Omron CX-Programmer project NewProject (CX-Programmer 9.73)

# PLC NewPLC1: CP2E-N N

## Global symbols (name address type ; comment)
0.00 BOOL  ; CR MASTER ON
0.01 BOOL  ; EMERGENCY STOP
0.02 BOOL  ; AUT: 1 / MAN: 0
0.03 BOOL  ; PB START AUTO
0.04 BOOL  ; PB RESET
0.05 BOOL  ; PB ROBOT RUN INSPECTION
0.06 BOOL  ; PB CLAMP
0.07 BOOL  ; PB UNCLAMP
0.08 BOOL  ; RS UNCLAMP 1
0.09 BOOL  ; RS UNCLAMP 2
0.10 BOOL  ; RS CLAMP 1
0.11 BOOL  ; RS CLAMP 2
100.00 BOOL  ; CR SOL CLAMP
100.01 BOOL  ; CR SOL UNCLAMP
100.02 BOOL  ; LAMP PLC RUN
100.03 BOOL  ; LAMP FAULT & TL RED
100.04 BOOL  ; LAMP HOMEPOST & TL GREEN
100.05 BOOL  ; LAMP AUTO RUN & TL YELLOW
100.06 BOOL  ; BUZZER
100.07 BOOL  ; LAMP ROBOT RUN
101.00 BOOL  ; TL INSPECTION OK
101.01 BOOL  ; TL INSPECTION NG
101.02 BOOL  ; TL INSPECTION RUN
10.00 BOOL  ; MASTER ON
10.01 BOOL  ; MASTER OFF
10.02 BOOL  ; MANUAL MODE CONFIRM
10.03 BOOL  ; AUTO MODE CONFIRM
10.04 BOOL  ; FAULT CONFIRM
10.05 BOOL  ; ROBOT ERROR
1.00 BOOL  ; PHS AGV
30.00 BOOL  ; IR CR UNCLAMP
30.01 BOOL  ; IR CR CLAMP
50.00 BOOL  ; AUTO UNCLAMP HOMING
50.01 BOOL  ; AUTO CLAMP
50.02 BOOL  ; AUTO ROBOT START INSPECTION
90.00 BOOL  ; MAN UNCLAMP
90.01 BOOL  ; MAN CLAMP
90.02 BOOL  ; MAN ROBOT START INSPECTION
T000 BOOL  ; DELAY RESET SEQ
T001 BOOL  ; DELAY AGV IN
W1 CHANNEL  ; ROBOT STATE
W2 CHANNEL  ; INSPECTION RESULT
W3 CHANNEL  ; ROBOT ERROR STATUS
W4 CHANNEL  ; ROBOT PROJECT STATUS
W5 CHANNEL  ; PLC ON STATUS
W6 CHANNEL  ; FLAG BARCODE FAIL

## Program NewProgram1 (cyclic task 0)

### Section MAIN_PROGRAM

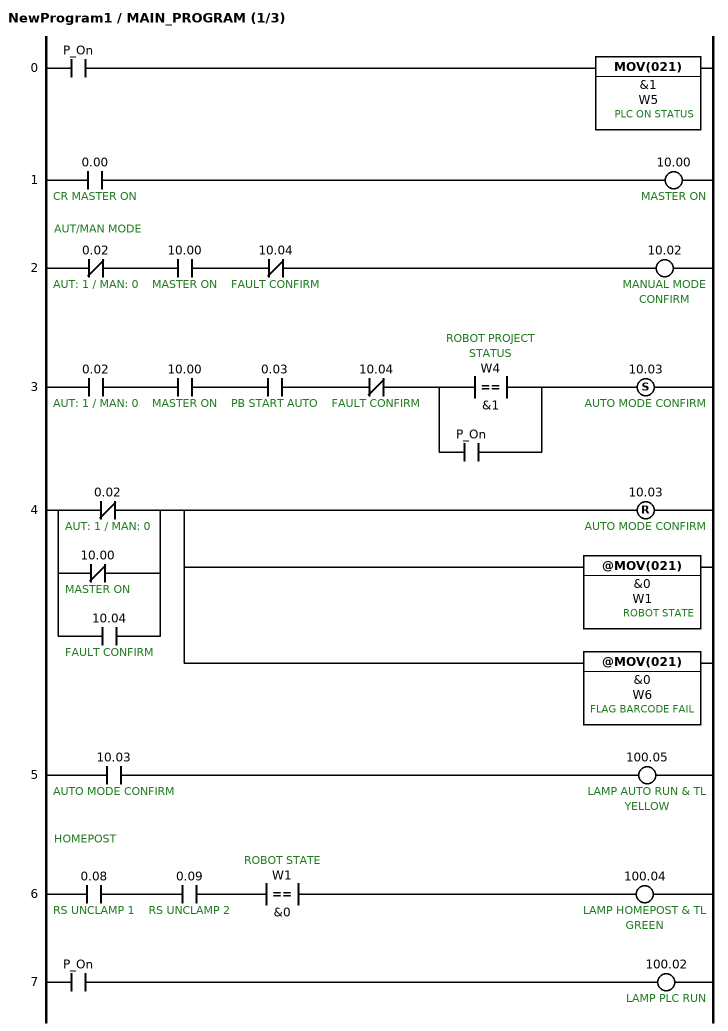
; rung 0
LD P_On
MOV(021) &1 W5  ; PLC ON STATUS
; rung 1
LD 0.00  ; CR MASTER ON
OUT 10.00  ; MASTER ON
; rung 2: AUT/MAN MODE
LDNOT 0.02  ; AUT: 1 / MAN: 0
AND 10.00  ; MASTER ON
ANDNOT 10.04  ; FAULT CONFIRM
OUT 10.02  ; MANUAL MODE CONFIRM
; rung 3
LD 0.02  ; AUT: 1 / MAN: 0
AND 10.00  ; MASTER ON
AND 0.03  ; PB START AUTO
ANDNOT 10.04  ; FAULT CONFIRM
LD=(300) W4 &1  ; ROBOT PROJECT STATUS
OR P_On
ANDLD
SET 10.03  ; AUTO MODE CONFIRM
; rung 4
LDNOT 0.02  ; AUT: 1 / MAN: 0
ORNOT 10.00  ; MASTER ON
OR 10.04  ; FAULT CONFIRM
RSET 10.03  ; AUTO MODE CONFIRM
@MOV(021) &0 W1  ; ROBOT STATE
@MOV(021) &0 W6  ; FLAG BARCODE FAIL
; rung 5
LD 10.03  ; AUTO MODE CONFIRM
OUT 100.05  ; LAMP AUTO RUN & TL YELLOW
; rung 6: HOMEPOST
LD 0.08  ; RS UNCLAMP 1
AND 0.09  ; RS UNCLAMP 2
AND=(300) W1 &0  ; ROBOT STATE
OUT 100.04  ; LAMP HOMEPOST & TL GREEN
; rung 7
LD P_On
OUT 100.02  ; LAMP PLC RUN

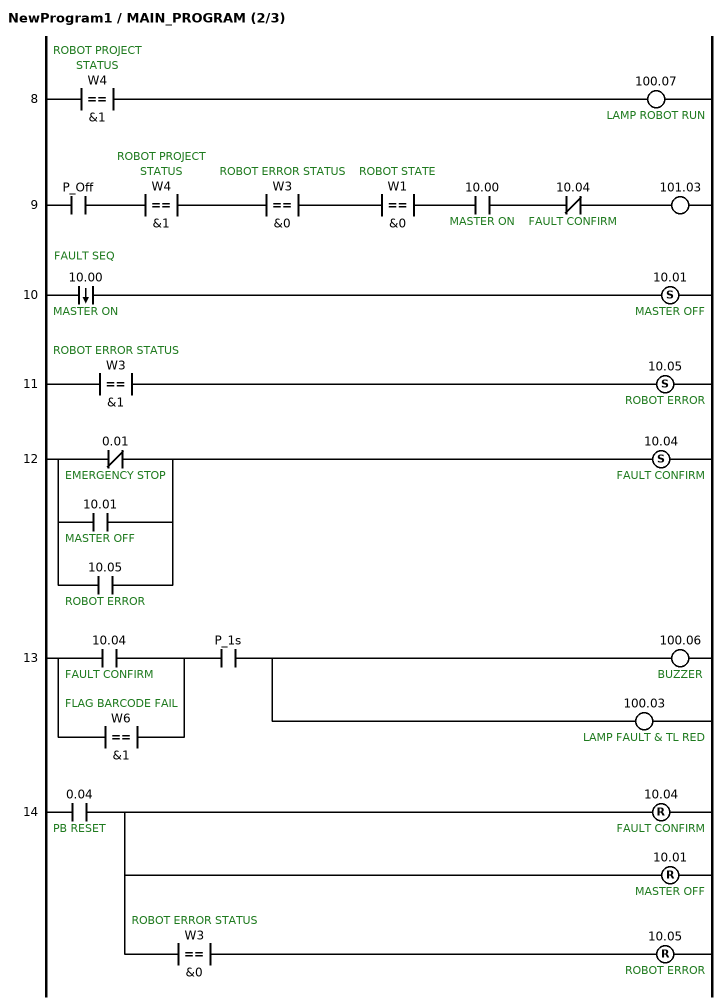
; rung 8
LD=(300) W4 &1  ; ROBOT PROJECT STATUS
OUT 100.07  ; LAMP ROBOT RUN
; rung 9
LD P_Off
AND=(300) W4 &1  ; ROBOT PROJECT STATUS
AND=(300) W3 &0  ; ROBOT ERROR STATUS
AND=(300) W1 &0  ; ROBOT STATE
AND 10.00  ; MASTER ON
ANDNOT 10.04  ; FAULT CONFIRM
OUT 101.03
; rung 10: FAULT SEQ
%LD 10.00  ; MASTER ON
SET 10.01  ; MASTER OFF
; rung 11
LD=(300) W3 &1  ; ROBOT ERROR STATUS
SET 10.05  ; ROBOT ERROR
; rung 12
LDNOT 0.01  ; EMERGENCY STOP
OR 10.01  ; MASTER OFF
OR 10.05  ; ROBOT ERROR
SET 10.04  ; FAULT CONFIRM
; rung 13
LD 10.04  ; FAULT CONFIRM
OR=(300) W6 &1  ; FLAG BARCODE FAIL
AND P_1s
OUT 100.06  ; BUZZER
OUT 100.03  ; LAMP FAULT & TL RED
; rung 14
LD 0.04  ; PB RESET
RSET 10.04  ; FAULT CONFIRM
RSET 10.01  ; MASTER OFF
AND=(300) W3 &0  ; ROBOT ERROR STATUS
RSET 10.05  ; ROBOT ERROR

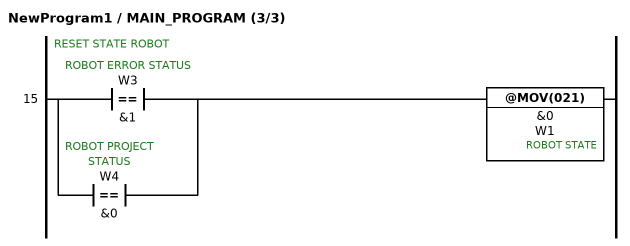
; rung 15: RESET STATE ROBOT
LD=(300) W3 &1  ; ROBOT ERROR STATUS
OR=(300) W4 &0  ; ROBOT PROJECT STATUS
@MOV(021) &0 W1  ; ROBOT STATE

### Section MANUAL

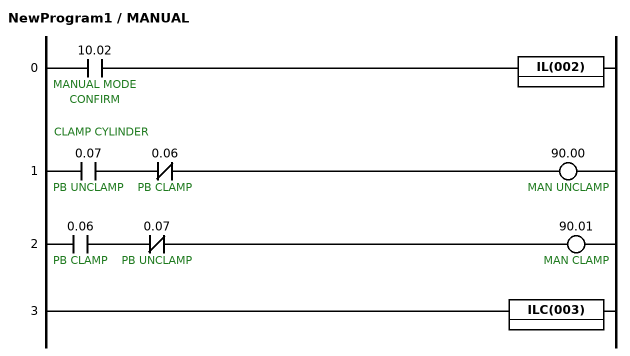
; rung 0
LD 10.02  ; MANUAL MODE CONFIRM
IL(002)
; rung 1: CLAMP CYLINDER
LD 0.07  ; PB UNCLAMP
ANDNOT 0.06  ; PB CLAMP
OUT 90.00  ; MAN UNCLAMP
; rung 2
LD 0.06  ; PB CLAMP
ANDNOT 0.07  ; PB UNCLAMP
OUT 90.01  ; MAN CLAMP
; rung 3
ILC(003)

### Section AUTO

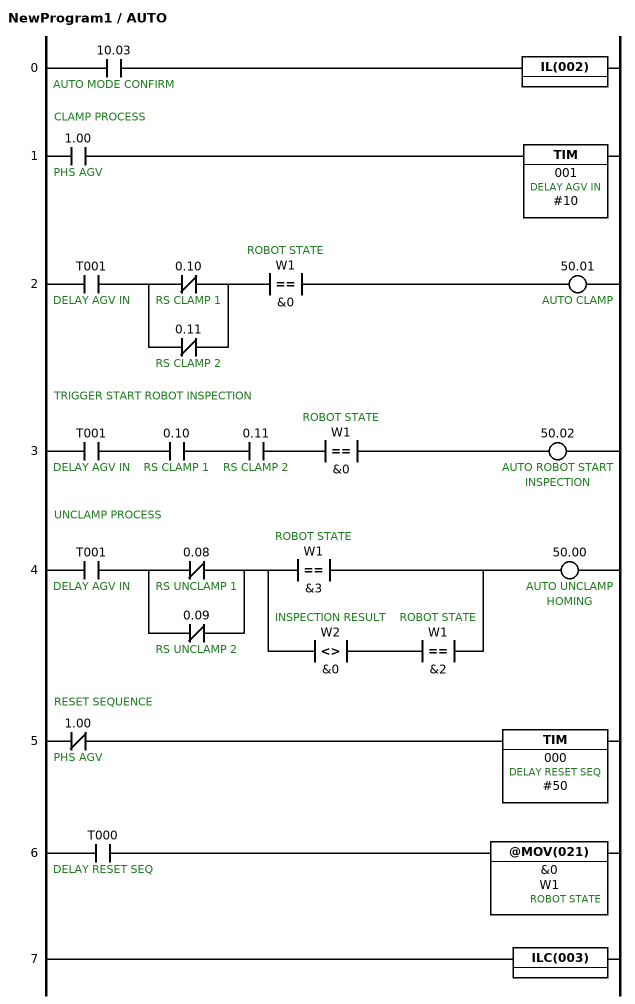
; rung 0
LD 10.03  ; AUTO MODE CONFIRM
IL(002)
; rung 1: CLAMP PROCESS
LD 1.00  ; PHS AGV
TIM 001 #10  ; DELAY AGV IN
; rung 2
LD T001  ; DELAY AGV IN
LDNOT 0.10  ; RS CLAMP 1
ORNOT 0.11  ; RS CLAMP 2
ANDLD
AND=(300) W1 &0  ; ROBOT STATE
OUT 50.01  ; AUTO CLAMP
; rung 3: TRIGGER START ROBOT INSPECTION
LD T001  ; DELAY AGV IN
AND 0.10  ; RS CLAMP 1
AND 0.11  ; RS CLAMP 2
AND=(300) W1 &0  ; ROBOT STATE
OUT 50.02  ; AUTO ROBOT START INSPECTION
; rung 4: UNCLAMP PROCESS
LD T001  ; DELAY AGV IN
LDNOT 0.08  ; RS UNCLAMP 1
ORNOT 0.09  ; RS UNCLAMP 2
ANDLD
LD=(300) W1 &3  ; ROBOT STATE
LD<>(305) W2 &0  ; INSPECTION RESULT
AND=(300) W1 &2  ; ROBOT STATE
ORLD
ANDLD
OUT 50.00  ; AUTO UNCLAMP HOMING
; rung 5: RESET SEQUENCE
LDNOT 1.00  ; PHS AGV
TIM 000 #50  ; DELAY RESET SEQ
; rung 6
LD T000  ; DELAY RESET SEQ
@MOV(021) &0 W1  ; ROBOT STATE
; rung 7
ILC(003)

### Section OUTPUT

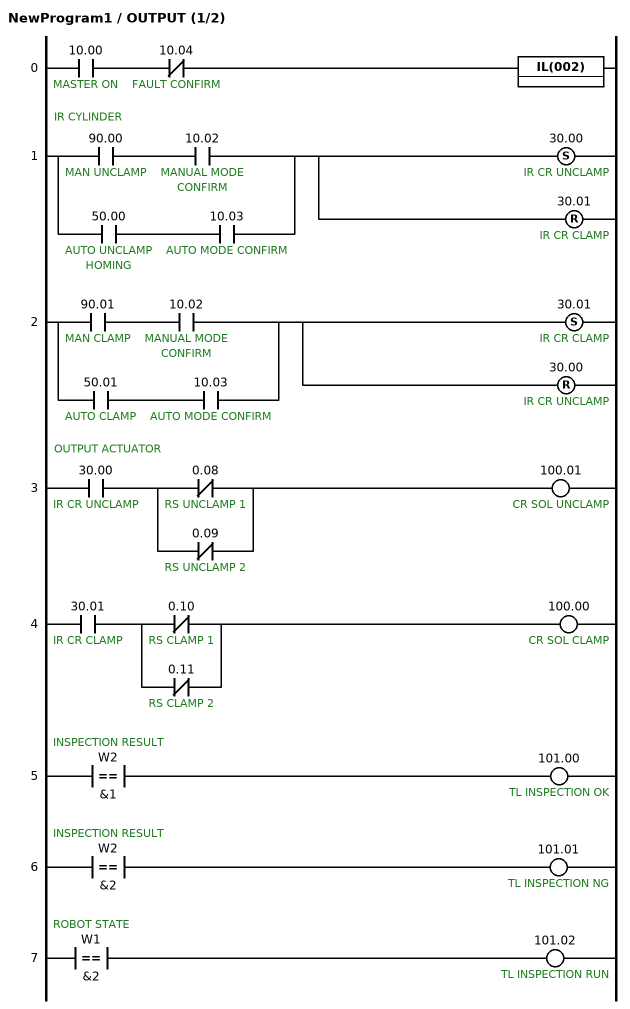
; rung 0
LD 10.00  ; MASTER ON
ANDNOT 10.04  ; FAULT CONFIRM
IL(002)
; rung 1: IR CYLINDER
LD 90.00  ; MAN UNCLAMP
AND 10.02  ; MANUAL MODE CONFIRM
LD 50.00  ; AUTO UNCLAMP HOMING
AND 10.03  ; AUTO MODE CONFIRM
ORLD
SET 30.00  ; IR CR UNCLAMP
RSET 30.01  ; IR CR CLAMP
; rung 2
LD 90.01  ; MAN CLAMP
AND 10.02  ; MANUAL MODE CONFIRM
LD 50.01  ; AUTO CLAMP
AND 10.03  ; AUTO MODE CONFIRM
ORLD
SET 30.01  ; IR CR CLAMP
RSET 30.00  ; IR CR UNCLAMP
; rung 3: OUTPUT ACTUATOR
LD 30.00  ; IR CR UNCLAMP
LDNOT 0.08  ; RS UNCLAMP 1
ORNOT 0.09  ; RS UNCLAMP 2
ANDLD
OUT 100.01  ; CR SOL UNCLAMP
; rung 4
LD 30.01  ; IR CR CLAMP
LDNOT 0.10  ; RS CLAMP 1
ORNOT 0.11  ; RS CLAMP 2
ANDLD
OUT 100.00  ; CR SOL CLAMP
; rung 5
LD=(300) W2 &1  ; INSPECTION RESULT
OUT 101.00  ; TL INSPECTION OK
; rung 6
LD=(300) W2 &2  ; INSPECTION RESULT
OUT 101.01  ; TL INSPECTION NG
; rung 7
LD=(300) W1 &2  ; ROBOT STATE
OUT 101.02  ; TL INSPECTION RUN

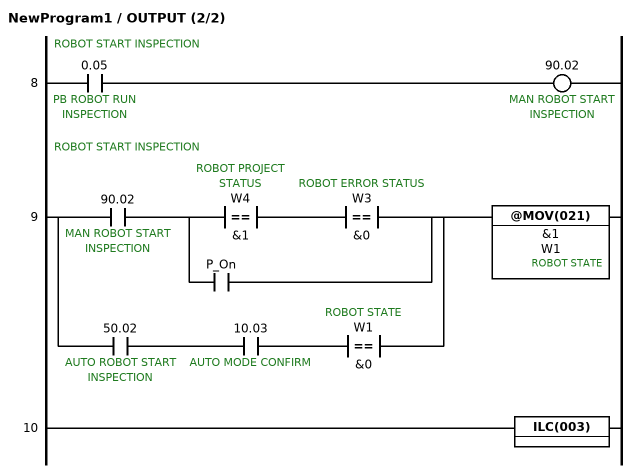
; rung 8: ROBOT START INSPECTION
LD 0.05  ; PB ROBOT RUN INSPECTION
OUT 90.02  ; MAN ROBOT START INSPECTION
; rung 9: ROBOT START INSPECTION
LD 90.02  ; MAN ROBOT START INSPECTION
LD=(300) W4 &1  ; ROBOT PROJECT STATUS
AND=(300) W3 &0  ; ROBOT ERROR STATUS
OR P_On
ANDLD
LD 50.02  ; AUTO ROBOT START INSPECTION
AND 10.03  ; AUTO MODE CONFIRM
AND=(300) W1 &0  ; ROBOT STATE
ORLD
@MOV(021) &1 W1  ; ROBOT STATE
; rung 10
ILC(003)

### Section END
; rung 0
END(001)